// TIA Portal V19 export
TYPE "C402_VAR_IF_SBO_TYPIC"
   STRUCT
      STS_BEZ_OPEN { ExternalAccessible := 'False'; ExternalVisible := 'False'; ExternalWritable := 'False'} : Bool;   // TRUE = Afsluitboom bezig met beweging openen
      STS_BEZ_TOE { ExternalAccessible := 'False'; ExternalVisible := 'False'; ExternalWritable := 'False'} : Bool;   // TRUE = Afsluitboom bezig met beweging sluiten
      STS_OPEN { ExternalAccessible := 'False'; ExternalVisible := 'False'; ExternalWritable := 'False'} : Bool;   // TRUE = Afsluitboom op stand Open
      STS_TOE { ExternalAccessible := 'False'; ExternalVisible := 'False'; ExternalWritable := 'False'} : Bool;   // TRUE = Afsluitboom op stand Dicht
      STS_STOP { ExternalAccessible := 'False'; ExternalVisible := 'False'; ExternalWritable := 'False'} : Bool;   // TRUE = Afsluitboom niet op een eindpositie en niet in beweging
      BMO_HAND { ExternalAccessible := 'False'; ExternalVisible := 'False'; ExternalWritable := 'False'} : Bool;   // TRUE = Afsluitboom in hand geschakeld / FALSE = niet in hand
      STS_VKL_OK { ExternalAccessible := 'False'; ExternalVisible := 'False'; ExternalWritable := 'False'} : Bool;   // TRUE = Verkeerslichten op Rood (voorwaarde voor sluiten)
      STS_NDS_OK { ExternalAccessible := 'False'; ExternalVisible := 'False'; ExternalWritable := 'False'} : Bool;   // TRUE = Geen noodstop (voorwaarde voor beweging)
      STS_LUS_OK { ExternalAccessible := 'False'; ExternalVisible := 'False'; ExternalWritable := 'False'} : Bool;   // TRUE = Detectielus(sen) OK (geen obstakel gedetecteerd voor sluiten)
      EXT_AUT { ExternalAccessible := 'False'; ExternalVisible := 'False'; ExternalWritable := 'False'} : Bool;   // Externe (hoofd) beveiliging aangesproken
      EXT_HW { ExternalAccessible := 'False'; ExternalVisible := 'False'; ExternalWritable := 'False'} : Bool;   // Sturings hardware (PLC) in storing
      EXT_STO { ExternalAccessible := 'False'; ExternalVisible := 'False'; ExternalWritable := 'False'} : Bool;   // Externe storing aanwezig
      LUS1_STS { ExternalAccessible := 'False'; ExternalVisible := 'False'; ExternalWritable := 'False'} : Bool;   // Detectie voertuig door lus 1 (1 = detectie)
      LUS2_STS { ExternalAccessible := 'False'; ExternalVisible := 'False'; ExternalWritable := 'False'} : Bool;   // Detectie voertuig door lus 2 (1 = detectie)
      LUS3_STS { ExternalAccessible := 'False'; ExternalVisible := 'False'; ExternalWritable := 'False'} : Bool;   // Detectie voertuig door lus 3 (1 = detectie)
      LUS4_STS { ExternalAccessible := 'False'; ExternalVisible := 'False'; ExternalWritable := 'False'} : Bool;   // Detectie voertuig door lus 3 (1 = detectie)
      STO { ExternalAccessible := 'False'; ExternalVisible := 'False'; ExternalWritable := 'False'} : Struct   // Opsomming van alle storingen
         A001 : Bool;   // Beveiliging aangesproken
         A002 : Bool;   // Storing van de detector van lus 1
         A003 : Bool;   // Storing van de detector van lus 2
         A004 : Bool;   // Storing van de detector van lus 3
         A005 : Bool;   // Storing van de detector van lus 4
         A006 : Bool;   // Storing van de motorsturing
         A007 : Bool;   // Storing motorbeveiliging
         AT01 : Bool;   // Terugmelding Open niet tijdig bereikt
         AT02 : Bool;   // Terugmelding Dicht niet tijdig bereikt
         AT03 : Bool;   // Terugmeldingen Open en Dicht tegelijkertijd
         AT04 : Bool;   // Terugmelding Open weggevallen
         AT05 : Bool;   // Terugmelding Dicht weggevallen
         M001 : Bool;   // Werkschakelaar uitgeschakeld
         M002 : Bool;   // Mechanische handbediening uitgenomen
      END_STRUCT;
   END_STRUCT;
END_TYPE
